% RSLogix 500 project CLOCK OPERATION CONTINUOS_BAK021.RSS, saved by version 8.30.00.16 %
PROJECT "UNTITLED"    % processor: Bul.1763 MicroLogix 1100 Series B %

PROGRAM FILES
  LAD 2   10 rungs

DATA FILES
  O0 OUTPUT  4 elements
  I1 INPUT  6 elements
  S2 STATUS  66 elements
  B3 BINARY  2 elements
  T4 TIMER  1 elements
  C5 COUNTER  3 elements
  R6 CONTROL  1 elements
  N7 INTEGER  3 elements
  F8 FLOAT  1 elements

LADDER 2
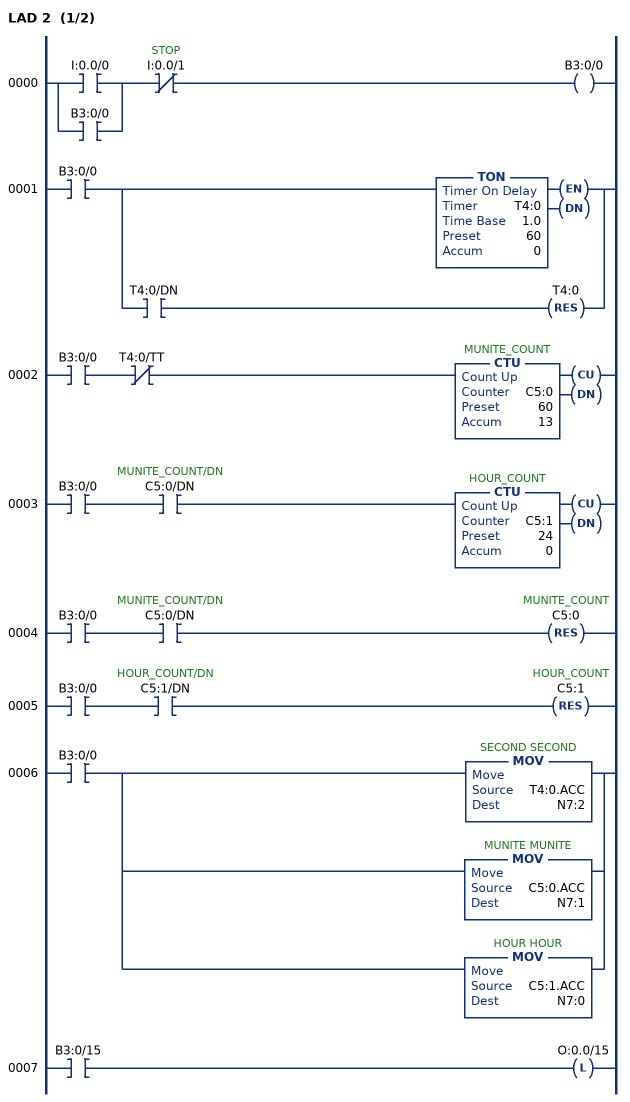
% Rung: 0 %
SOR BST XIC I:0.0/0 NXB XIC B3:0/0 BND XIO I:0.0/1 OTE B3:0/0 EOR
%   I:0.0/1  STOP %
% Rung: 1 %
SOR XIC B3:0/0 BST TON T4:0 1.0 60 0 NXB XIC T4:0/DN RES T4:0 BND EOR
% Rung: 2 %
SOR XIC B3:0/0 XIO T4:0/TT CTU C5:0 60 13 EOR
%   C5:0  MUNITE_COUNT %
% Rung: 3 %
SOR XIC B3:0/0 XIC C5:0/DN CTU C5:1 24 0 EOR
%   C5:0  MUNITE_COUNT %
%   C5:1  HOUR_COUNT %
% Rung: 4 %
SOR XIC B3:0/0 XIC C5:0/DN RES C5:0 EOR
%   C5:0  MUNITE_COUNT %
% Rung: 5 %
SOR XIC B3:0/0 XIC C5:1/DN RES C5:1 EOR
%   C5:1  HOUR_COUNT %
% Rung: 6 %
SOR XIC B3:0/0 BST MOV T4:0.ACC N7:2 NXB MOV C5:0.ACC N7:1 NXB MOV C5:1.ACC N7:0 BND EOR
%   N7:2  SECOND  "SECOND" %
%   C5:0  MUNITE_COUNT %
%   N7:1  MUNITE  "MUNITE" %
%   C5:1  HOUR_COUNT %
%   N7:0  HOUR  "HOUR" %
% Rung: 7 %
SOR XIC B3:0/15 OTL O:0.0/15 EOR

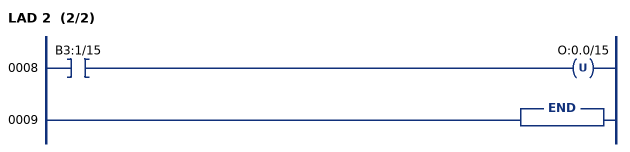
% Rung: 8 %
SOR XIC B3:1/15 OTU O:0.0/15 EOR
% Rung: 9 %
SOR END EOR

OTHER DOCUMENTED ADDRESSES
  I:0  PUSH  "START"

DATA TABLE (non-zero values as saved)
DATA B3
% B3:0 % 0X0002 0X0000
DATA T4
% .PRE .ACC %
% T4:0 % 60 0
DATA C5
% .PRE .ACC %
% C5:0 % 60 13
% C5:1 % 24 0
DATA N7
% N7:0 % 0 13 5
